// TIA Portal V19 export
TYPE "M0940_PIDInterface"
   STRUCT
      PV : Real;
      SP : Real;
      EngUnitsMin : Real;
      EngUnitsMax : Real;
      P : Real;
      I : Time;
      D : Time;
   END_STRUCT;
END_TYPE
